(* IEC 61131-3 sources: AXOpen/src/timers/src, 2 files *)

(* ---- OffDelay.st ---- *)
USING AXOpen.Core;

NAMESPACE AXOpen.Timers

    CLASS OffDelayContext
        VAR PUBLIC
            output : BOOL;
            elapsedTime : LTIME;
        END_VAR

        VAR PRIVATE
          _startTime : LDATE_AND_TIME;
          _previousSignalStatus : BOOL;
          _currentTimeDiff : LTIME;
          _isCounting : BOOL;

        END_VAR

        /// When IN is TRUE, Q is TRUE and ET is 0.
        /// As soon as IN becomes FALSE, the time will begin to be counted in milliseconds in ET until its value is equal to that of PT.
        /// It will then remain constant.
        /// Q is FALSE when IN is FALSE and ET is equal to PT.
        /// Otherwise it is TRUE.
        /// Thus, Q has a falling edge when the time indicated in PT in milliseconds has run out.

        ///<summary>
        /// OffDelay timer, which output it FALSE when time delay is counted, otherwise always returns TRUE.
        /// Counting of timer start on FALLING edge.
        ///</summary>
        METHOD PUBLIC OffDelay : BOOL
            VAR_INPUT
                Context : IAxoContext;
                inSignal : BOOL;
                TimeDelay : LTIME;
            END_VAR

            IF(Context = NULL) THEN RETURN; END_IF;

            // if input signal is off and previous signal was off, no edge detected, return output false
            IF(NOT inSignal AND NOT THIS._previousSignalStatus) THEN
                OffDelay := FALSE;
                output := OffDelay;
                THIS._previousSignalStatus := inSignal;
                RETURN;
            END_IF;

            // RISING EDGE detected, set output to true
            // if inSignal is true, and previous is false, set output to true
            // restore timer on rising edge
            IF(inSignal AND NOT THIS._previousSignalStatus) THEN
                THIS.Restore();
                OffDelay := TRUE;
                output := OffDelay;
                THIS._previousSignalStatus := inSignal;
                RETURN;
            END_IF;

           // FALLING EDGE  detected start timer counting
           // start computing on falling edge (if actual signal is false, but previous was true)
            IF(NOT inSignal AND THIS._previousSignalStatus) THEN
                THIS._startTime := Context.GetRtc().NowUTC();
                _isCounting := TRUE;
            END_IF;

             // if timer is counting, compute difference and watch for end of timer
            IF(THIS._isCounting) THEN
                _currentTimeDiff := Context.GetRtc().NowUTC() - THIS._startTime ;
                // if timer passed, set output to false
                OffDelay := NOT (_currentTimeDiff >= TimeDelay);
                output := OffDelay;
                elapsedTime :=  _currentTimeDiff;
                THIS._previousSignalStatus := inSignal;

            ELSE
                // here timer is not counting, therefore output will be set to true
                // I get here, when previousSignal was true, and actual signal is still true
                OffDelay := TRUE;
                output := OffDelay;
                elapsedTime :=  LTIME#0s;
                THIS._previousSignalStatus := inSignal;
            END_IF;

        END_METHOD

        // LDT#1980-01-23-13:14:33.123456
        // LTIME#13:14:3.45;
        METHOD PUBLIC Restore
            //_startTime := LDT#0;
            _isCounting := FALSE;

            _previousSignalStatus := FALSE;
            _currentTimeDiff := LTIME#0s;
            _startTime := LDATE_AND_TIME#1970-01-01-00:00:00.000;

        END_METHOD

    END_CLASS
END_NAMESPACE

(* ---- OnDelay.st ---- *)
USING AXOpen.Core;

NAMESPACE AXOpen.Timers

    CLASS OnDelayContext
        VAR PUBLIC
            output : BOOL;
            elapsedTime : LTIME;
        END_VAR

        VAR PRIVATE
          _startTime : LDATE_AND_TIME;
          _previousSignalStatus : BOOL;
          _currentTimeDiff : LTIME;

        END_VAR

        /// If IN is FALSE, Q is FALSE and ET is 0.
        /// As soon as IN becomes TRUE, the time will begin to be counted in milliseconds in ET until its value is equal to PT.
        /// It will then remain constant. Q is TRUE when IN is TRUE and ET is equal to PT.
        /// Otherwise it is FALSE.
        /// Thus, Q has a rising edge when the time indicated in PT in milliseconds has run out.

        ///<summary>
        /// OnDelay timer, which output is TRUE when time delay is counted, otherwise always returns FALSE.
        /// Counting of timer start on RISING edge.
        ///</summary>
        METHOD PUBLIC OnDelay : BOOL
            VAR_INPUT
                Context : IAxoContext;
                inSignal : BOOL;
                TimeDelay : LTIME;
            END_VAR

            IF(Context = NULL) THEN RETURN; END_IF;

            // beggining, if all is turn off, return false
            IF(NOT inSignal AND NOT THIS._previousSignalStatus) THEN
                OnDelay := FALSE;
                output := OnDelay;
                elapsedTime := LTIME#0s;
                RETURN;
            END_IF;

            // start counting on RISING edge
            // start counting when inputSignal is true and previous signal was not set
            IF(inSignal AND NOT THIS._previousSignalStatus) THEN
                THIS._startTime := Context.GetRtc().NowUTC();
            END_IF;

            // FALLING edge detected
            // if input signal is turned off and previous signal was true, that means output must by false, we do not need to compute time
            // let's afterwards restore timer to default values
            IF(NOT inSignal AND THIS._previousSignalStatus) THEN
                THIS.Restore();
                THIS._previousSignalStatus := inSignal;
                OnDelay := FALSE;
                output := OnDelay;
                elapsedTime := _currentTimeDiff;

                RETURN;
            END_IF;

            _currentTimeDiff := Context.GetRtc().NowUTC() - THIS._startTime ;
            OnDelay := _currentTimeDiff >= TimeDelay;
            output := OnDelay;
            elapsedTime :=  _currentTimeDiff;
            THIS._previousSignalStatus := inSignal;

        END_METHOD

        METHOD PUBLIC Restore
            _previousSignalStatus := FALSE;
            _currentTimeDiff := LTIME#0s;
            //_startTime := LDATE_AND_TIME#1970-01-01-00:00:00.000;
        END_METHOD

        //LDT#1980-01-23-13:14:33.123456
        // LTIME#13:14:3.45;
        // METHOD PUBLIC Delay : BOOL
        //     VAR_INPUT
        //         Parent : IAxoObject;
        //         Signal : BOOL;
        //         TimeDelay : LTIME;
        //     END_VAR

        //     IF(Parent = NULL) THEN RETURN; END_IF;

        //     IF(Signal AND NOT THIS._previousSignalStatus) THEN
        //         THIS._startTime := Parent.GetContext().GetRtc().NowUTC();
        //     END_IF;

        //     Delay := (THIS._startTime - Parent.GetContext().GetRtc().NowUTC()) >= TimeDelay;
        //     output := Delay;
        //     THIS._previousSignalStatus := Signal;
        // END_METHOD

        // CLASS OnDelay
    //     VAR
    //         _timeBase : LINT := LINT#10;
    //         _timeBaseTickCounter : INT;
    //         _previousSignalStatus : BOOL;
    //         _timeasint : LINT;
    //     END_VAR

    //     METHOD PUBLIC Delay : BOOL
    //         VAR_INPUT
    //             Signal : BOOL;
    //             TimeDelay : TIME;
    //         END_VAR

    //         IF(Signal AND NOT _previousSignalStatus) THEN
    //             _timeasint := TO_LINT(TimeDelay);
    //             _timeBaseTickCounter := 0;
    //         END_IF;

    //         _timeBaseTickCounter := _timeBaseTickCounter + 1;
    //         Delay := TO_TIME((_timeBaseTickCounter * _timeBase)) >= TimeDelay;

    //         _previousSignalStatus := Signal;
    //     END_METHOD

    // END_CLASS
    END_CLASS
END_NAMESPACE
